function_block FB_Syntax_ExST var nI      : int; nSum  : int; bFlag   : bool; rRef        : reference to int; nTarget : int; end_var

if (nI <> 0) and_then (nSum > 0) or bFlag then
nSum := nSum + 1;
end_if


for nI := 1 to 5 do if nI mod 2 = 0 then continue; end_if
nSum := nSum + nI;
end_for


JMP _skip;
nSum := -1;
_skip:


rRef REF= nTarget;
rRef := 42;

END_FUNCTION_BLOCK

(* stored: Version 1.1.0.1, ProductVersion 3.1.4024.16
   POU FB_Syntax_ExST: Id {a9ca13e1-51a6-46c6-ba73-5a846c68aec3}, SpecialFunc None *)
